PROGRAM MAIN
VAR
	fbRead : ADSREAD;
	value : bool;
END_VAR

fbRead(
	NETID:= '5.58.198.104.1.2', 
	PORT:= 851, 
	IDXGRP:= 16#4020, 
	IDXOFFS:= 127, 
	LEN:= SIZEOF(value), 
	DESTADDR:= ADR(value), 
	READ:= , 
	TMOUT:= , 
	BUSY=> , 
	ERR=> , 
	ERRID=> );

END_PROGRAM

(* stored: Version 1.1.0.1, ProductVersion 3.1.4022.10
   POU MAIN: Id {1a75462b-9732-4735-b360-a17758a8c75a}, SpecialFunc None *)
